FUNCTION_BLOCK VIDEOWRITER (* openCV write video *)
  (* Version 1.0, AN, SWDC RTSoft *)
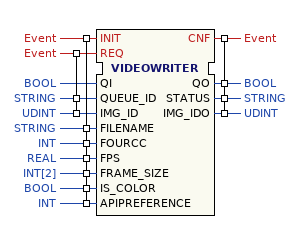
  EVENT_INPUT
    INIT WITH FILENAME, FOURCC, FPS, FRAME_SIZE, IS_COLOR, APIPREFERENCE;
    REQ WITH QUEUE_ID, IMG_ID;
  END_EVENT
  EVENT_OUTPUT
    CNF WITH QO, STATUS, IMG_IDO;
  END_EVENT
  VAR_INPUT
    QI : BOOL;
    QUEUE_ID : STRING;
    IMG_ID : UDINT;
    FILENAME : STRING;
    FOURCC : INT;
    FPS : REAL;
    FRAME_SIZE : ARRAY [0..1] OF INT;
    IS_COLOR : BOOL;
    APIPREFERENCE : INT;
  END_VAR
  VAR_OUTPUT
    QO : BOOL;
    STATUS : STRING;
    IMG_IDO : UDINT;
  END_VAR
  (* Service APPLICATION/RESOURCE: Service Interface Function Block Type *)
END_FUNCTION_BLOCK
